{attribute 'linkalways'} 
{attribute 'no_explicit_call' := 'This FB is a CLASS and must be accessed using methods or properties'}
{attribute 'enable_dynamic_creation'}
FUNCTION_BLOCK Node_F_VN_PadImageBorder EXTENDS VisionNode
VAR
    ipSrcImage : _ITcVnImage;
    ipPaddedImage : _ITcVnImage;
    nTopBorder : _UDINT(0);
    nBottomBorder : _UDINT(0);
    nLeftBorder : _UDINT(0);
    nRightBorder : _UDINT(0);
    hrPrev : _HRESULT(S_OK);
	hresult : _HRESULT(S_OK);
END_VAR

METHOD PUBLIC  Clone : I_Node
VAR
	pNode : POINTER TO Node_F_VN_PadImageBorder;
END_VAR
pNode := __NEW(Node_F_VN_PadImageBorder);
Clone := pNode^;
END_METHOD

METHOD FB_init : BOOL
VAR_INPUT
	bInitRetains : BOOL; // if TRUE, the retain variables are initialized (warm start / cold start)
	bInCopyCode : BOOL;  // if TRUE, the instance afterwards gets moved into the copy code (online change)
END_VAR
AddInput('ipSrcImage', ipSrcImage);
AddParameter('nTopBorder', nTopBorder);
AddParameter('nBottomBorder', nBottomBorder);
AddParameter('nLeftBorder', nLeftBorder);
AddParameter('nRightBorder', nRightBorder);
AddInput('hrPrev', hrPrev);
AddOutput('ipPaddedImage', ipPaddedImage);
AddOutput('hresult',hresult);
END_METHOD

METHOD PROTECTED OnExecute
hresult.Value := F_VN_PadImageBorder(
    ipSrcImage := ipSrcImage.Value,
	ipPaddedImage := ipPaddedImage.Value,
    nTopBorder := nTopBorder.Value,
    nBottomBorder := nBottomBorder.Value,
    nLeftBorder := nLeftBorder.Value,
    nRightBorder := nRightBorder.Value,
	hrPrev:= hrPrev.Value);
END_METHOD

METHOD PUBLIC PreExecutionCheck
VAR_INPUT
	Check : I_PreExecutionChecks;
END_VAR
Check.IsTrue(ipSrcImage.IsValid, 'ipSrcImage must contain an image');
END_METHOD

END_FUNCTION_BLOCK

(* stored: Version 1.1.0.1, ProductVersion 3.1.4024.15
   POU Node_F_VN_PadImageBorder: Id {17dd5bc8-4942-0786-1bf5-8687bbcbc976}, SpecialFunc None
   Folder Constructor: Id {2a666cca-e194-0c2c-2606-ea7cb1d75e2e}
   Method Clone: Id {df0879b7-ac98-0a9e-0af0-a50856f79424}
   Method FB_init: Id {8714c7c6-d6c2-0217-2151-460f00cbf584}
   Method OnExecute: Id {10ca4504-b960-0d8e-0d78-0089290996a7}
   Method PreExecutionCheck: Id {c8a8c610-b7d6-0373-1bd9-f2c552719cba} *)
